(* PLC project rotary_plate_ring, Dassault Systèmes ControlBuild 2024x *)
(* stored: creationDateTime 2023-10-03T11:12:55-01:00 *)

(* This module simulates the behaviour of a rotary plate ring. It takes a rotation speed as input and can move actors and products that are in interaction. *)
FUNCTION_BLOCK equipment_library.rotary_plate_ring
  VAR_INPUT
    incShiftX : REAL := 0.0;
    incShiftZ : REAL := 0.0;
    incShiftY : REAL := 0.0;
  END_VAR
  VAR_INPUT
    rotationSpeed : REAL := 0.0;
  END_VAR
  VAR_OUTPUT
    angleRotationRad : REAL := 0.0;
    incRotation : REAL := 0.0;
    centerX : REAL := 0.0;
    centerY : REAL := 0.0;
    centerZ : REAL := 0.0;
    angleRotationDeg : REAL := 0.0;
  END_VAR
  VAR
    status_act_prod : DINT := 0;
    m11 : REAL := 1.0;
    m12 : REAL := 0.0;
    m13 : REAL := 0.0;
    m14 : REAL := 0.0;
    m21 : REAL := 0.0;
    m22 : REAL := 1.0;
    m23 : REAL := 0.0;
    m24 : REAL := 0.0;
    m31 : REAL := 0.0;
    m32 : REAL := 0.0;
    m33 : REAL := 1.0;
    m34 : REAL := 0.0;
    m41 : REAL := 0.0;
    m42 : REAL := 0.0;
    m43 : REAL := 0.0;
    m44 : REAL := 1.0;
    incrementRotation : REAL := 0.0;
  END_VAR
  VAR CONSTANT
    positionsRecalage : ARRAY[1..5] OF REAL := [0.0, 90.0, 180.0, 270.0, 360.0];
    deltaPos : REAL := 10.0;
  END_VAR
  VAR
    d_locking : BOOL := false;
    v_d_locking : REAL := 0.0;
    d_position : BOOL := false;
    v_d_position : REAL := 0.0;
  END_VAR


ACTION C_source_code:
/* ----------------------------------------------------------------	*/
/* Type : Model of Operative Behaviour					*/
/* Category :  Actors and Products						*/
/* Author : Dassault Systemes						*/
/* Update date : June 2018							*/
/* ----------------------------------------------------------------	*/
/* This module simulates the behaviour of a rotary plate ring.	*/
/* It takes a rotation speed as input and can move actors and		*/
/* products that are in interaction.					*/
/* ----------------------------------------------------------------	*/

/* ----------------------------------------------------------------	*/
/* Management of the rotation						*/
/* ----------------------------------------------------------------	*/
if (d_locking) 
	incrementRotation = 0;
else {
	/* Compute the increment of rotation according to the simulation clock	*/
	incrementRotation = rotationSpeed * (CLOCK_PERIOD/1000000.0) ;	
}

/* ----------------------------------------------------------------	*/
/* Request for updating the plate ring's position 			*/
/* ----------------------------------------------------------------	*/
if (d_position) {
	incrementRotation = v_d_position - getAngleZ(myself);
	d_position = 0;
}

/* ----------------------------------------------------------------	*/
/* Request for align the tipper in fixed position 			*/
/* ----------------------------------------------------------------	*/
if (rotationSpeed == 0.0) {
	CB_Int i;
	CB_Float currentAngle;
	currentAngle=getAngleZ(myself);  
	for (i=1; i<=5; i++) {
		if ((currentAngle- deltaPos < positionsRecalage(i)) && (currentAngle+ deltaPos > positionsRecalage(i))) {
			incrementRotation = positionsRecalage(i) - currentAngle;
			break;
		 }
	}
}
/* ----------------------------------------------------------------	*/
/* Rotation of the plate ring						*/
/* ----------------------------------------------------------------	*/
if (incrementRotation != 0.0)
	rotateCenterBy(myself, 0.0, 0.0, incrementRotation);

/* ----------------------------------------------------------------	*/
/* Compute the rotation angle in degrees and in radians		*/
/* ----------------------------------------------------------------	*/
angleRotationDeg = getAngleZ(myself);
angleRotationRad = angleRotationDeg * PI/180.0;


/* ----------------------------------------------------------------	*/
/* Shift the plate ring			    				*/
/* ----------------------------------------------------------------	*/
if (incShiftX != 0.0) moveXBy(myself, incShiftX);
if (incShiftY != 0.0) moveYBy(myself, incShiftY);
if (incShiftZ != 0.0) moveZBy(myself, incShiftZ);

/* ----------------------------------------------------------------	*/
/* Compute the rotation center of the plate ring			*/
/* ----------------------------------------------------------------	*/
centerX = getCenterX(myself);
centerY = getCenterY(myself);
centerZ = getCenterZ(myself);

/* ----------------------------------------------------------------	*/
/* Output of the rotation angle for rotated actors/products		*/
/* ----------------------------------------------------------------	*/
incRotation = incrementRotation;
END_ACTION

ACTION C_header:
#ifndef PI
#define PI 3.1415926535898
#endif
END_ACTION
END_FUNCTION_BLOCK
